TEXTLIST TL_Supply
  1 = 'fPwmCycleTime'
  2 = 'fPwmMinOnTime'
  3 = 'fPwmMaxOnTime'
  4 = 'fPwmMaxOnC'
  5 = 'fPwmMaxRampLoad'
  6 = 'fActSupplyLoad'
  7 = 'fActSupplyLoad'
  8 = 'fActSupplyCurrent'
  9 = 'fSupplyLoad'
  10 = 'fSupplyMatch'
   = ''
END_TEXTLIST

(* stored: Version 1.1.0.1, ProductVersion 3.1.4018.5
   TextList TL_Supply: Id {da378d31-91f8-4d8d-bebd-803b0943684b} *)
